Universal Robots PolyScope program: TP1_Q11G.urp

Program TP1_Q11G (installation=default directory=/home/ur/ursim-current/programs createdIn=5.9.4 lastSavedIn=5.13.1 robotSerialNumber=20195599999)
Calibrated DH parameters: a=[0, -0.425, -0.3922, 0, 0, 0]; d=[0.1625, 0, 0, 0.1333, 0.0997, 0.0996]; alpha=[1.570796, 0, 0, 1.570796, -1.570796, 0]; deltaTheta=[0, 0, 0, 0, 0, 0]
InitVariablesNode
BeforeStart
  Script file /home/ur/ursim-current/programs/TP1_Q1_BeforeStart.script
    | ### Definition des constantes ###
    | 
    | alpha = d2r(60)
    | 
    | # Position du robot (coord. homogene) lorsque beta = 90 deg
    | position = [0, -0.6, 0.3, 1]
    | 
    | # Transformation homogene entre la base et le support incline
    | H1 = [[sin(alpha),0,cos(alpha),0], [0,1,0,0], [-cos(alpha),0,sin(alpha),0], [0,0,0,1]]
    | H2 = [[0,1,0,0.7], [-1,0,0,0], [0,0,1,0], [0,0,0,1]]
    | H = H1*H2
    | 
    | # Variation de beta pour la loop
    | i = 0
    | DeltaBeta = 5
    | betaMin = 30
    | betaMax = 150
    | betaDeg = betaMin
Robot Program (runOnlyOnce=true)
  MoveJ speed 60 deg/s, acceleration 80 deg/s^2 (useActiveTCP=true) feature=Base
    Waypoint pose_ini: TCP in base x=-80.659 y=-681.405 z=687.2 mm, rx=1.5708 ry=0 rz=0 rad; joints [60, -90, 90, -180, -60, 180] deg; TCP offset x=0 y=0 z=175.5 mm, rx=0 ry=0 rz=0 rad
  Script file /home/ur/ursim-current/programs/TP1_Q1_OrientationG.script
    | ### Fonction permettant d'obtenir les invariants naturels a partir de alpha et beta ###
    | 
    | def Orientation(alpha, beta):
    | 
    | 	# --- Implementer les invariants naturels phi et e ici --- #
    | 	R10=[[0,-1,0], [1,0,0], [0,0,1]]
    | 	R21=[[sin(alpha),0,-cos(alpha)], [0,1,0], [cos(alpha),0,sin(alpha)]]
    | 
    | 	R32=[[cos(beta),0,-sin(beta)], [-sin(beta),0,-cos(beta)], [0,1,0]]
    | 	R30=R10*R21*R32
    | 	VECT=0.5*[R30[2,1] - R30[1,2]  , R30[0,2] - R30[2,0], R30[1,0] - R30[0,1]]
    | 	TR=R30[0,0]+ R30[1,1] + R30[2,2]
    | 	SINPHI=norm(VECT)
    | 	COSPHI=(TR-1)/2
    | 	phi = atan2(SINPHI,COSPHI)
    | 	e = VECT/norm(VECT)
    | 
    | 
    | 
    | 	# ------------ #
    | 
    | 	# Orientation de l'effecteur (axis-angle notation)
    | 	AxisAngle = phi*e
    | 	return AxisAngle
    | end
  Script file /home/ur/ursim-current/programs/TP1_Q1.script
    |     ### Programme principale : Loop sur les valeurs de beta ###
    | 
    |     while betaDeg <= betaMax:
    | 
    |             	beta = d2r(betaDeg)
    | 
    |             	# Position de l'effecteur
    |             	gamma = beta - 1.57
    |             	Q = [[cos(gamma),sin(gamma),0,0], [-sin(gamma),cos(gamma),0,0], [0,0,1,0], [0,0,0,1]]
    |             	positionNew = inv(H)*Q*H*position
    | 
    |             	# Orientation de l'effecteur
    |             	AxisAngle = Orientation(alpha, beta)
    |   	textmsg("AxisAngle",beta)
    | 	#writer.appendLine(textmsg("The axis angle"),beta)
    |             	# Pose de l'effecteur
    |             	pose = p[positionNew[0], positionNew[1], positionNew[2], AxisAngle[0], AxisAngle[1], AxisAngle[2]]
    | 
    |             	# Deplacement lineaire (tool-space)
    |             	movel(pose, a=0.2, v=0.05, t=0, r=0.01)
    | 
    |            	i = i+1
    |     	betaDeg = betaMin + DeltaBeta*i
    |     end
    |   end
    | end
